// TIA Portal project "FactoryIO_Template_S7-1200_V15_V17" (V17)
// Vorlageprojekt für das Buch mit Zielsystem S7-1200

(* hardware
DEVICE "S7-1200-Station_1"  S7-1200 Station
   slot 0: "Baugruppenträger_0"  Rack  V1.0
   slot 1: "PLC_1"  CPU 1211C DC/DC/DC  6ES7 211-1AE40-0XB0  V4.1
*)

// ===== PLC "PLC_1"  CPU 1211C DC/DC/DC =====

VAR_GLOBAL   // PLC tag table "Inputs"
   "start_button" AT %I0.0 : Bool;
   "stop_button" AT %I0.1 : Bool;
   "reset_counters_button" AT %I0.2 : Bool;
   "blue_vision_sensor" AT %I0.3 : Bool;
   "green_vision_sensor" AT %I0.4 : Bool;
   "blue_count_sensor" AT %I0.5 : Bool;
   "green_count_sensor" AT %I0.6 : Bool;
   "metal_count_sensor" AT %I0.7 : Bool;
   "safety_door" AT %I1.0 : Bool;
   "emergency_stop" AT %I1.1 : Bool;
END_VAR

VAR_GLOBAL   // PLC tag table "Outputs"
   "main_conveyor" AT %Q0.0 : Bool;
   "conveyor1(blue)" AT %Q0.1 : Bool;
   "conveyor2(green)" AT %Q0.2 : Bool;
   "conveyor3(else)" AT %Q0.3 : Bool;
   "curved_conveyor" AT %Q0.4 : Bool;
   "blue_pusher" AT %Q0.5 : Bool;
   "green_pusher" AT %Q0.6 : Bool;
   "emitter" AT %Q0.7 : Bool;
   "blue_dispatch_pusher" AT %Q1.0 : Bool;
   "blue_reset" AT %Q1.1 : Bool;
   "green_dispatch_pusher" AT %Q1.2 : Bool;
   "green_reset" AT %Q1.3 : Bool;
   "metal_dispatch_pusher" AT %Q1.4 : Bool;
   "metal_reset" AT %Q1.5 : Bool;
   "alarm_siren" AT %Q1.6 : Bool;
   "warning_light" AT %Q1.7 : Bool;
   "start_light" AT %Q2.0 : Bool;
   "stop_light" AT %Q2.1 : Bool;
   "factoryIo_reset" AT %Q2.2 : Bool;
END_VAR

VAR_GLOBAL   // PLC tag table "Memory"
   "system" AT %M0.0 : Bool;
   "blue_current_value" AT %MW1 : Word;
   "green_current_value" AT %MW2 : Word;
   "metal_current_value" AT %MW3 : Word;
END_VAR

// folder: System blocks/Program resources

DATA_BLOCK "blue_counter"   // DB1
{ S7_Optimized_Access := 'TRUE' }
AUTHOR : Simatic
FAMILY : IEC
NAME : CNTR
VERSION : 1.0
// stored: InstanceOfName IEC_COUNTER
"IEC_COUNTER"
BEGIN
END_DATA_BLOCK

DATA_BLOCK "blue_delay"   // DB2
{ S7_Optimized_Access := 'TRUE' }
AUTHOR : Simatic
FAMILY : IEC
NAME : IEC_TMR
VERSION : 1.0
// stored: InstanceOfName IEC_TIMER
"IEC_TIMER"
BEGIN
END_DATA_BLOCK

DATA_BLOCK "IEC_Timer_0_DB"   // DB3
{ S7_Optimized_Access := 'TRUE' }
AUTHOR : Simatic
FAMILY : IEC
NAME : IEC_TMR
VERSION : 1.0
// stored: InstanceOfName IEC_TIMER
"IEC_TIMER"
BEGIN
END_DATA_BLOCK

DATA_BLOCK "green_counter"   // DB4
{ S7_Optimized_Access := 'TRUE' }
AUTHOR : Simatic
FAMILY : IEC
NAME : CNTR
VERSION : 1.0
// stored: InstanceOfName IEC_COUNTER
"IEC_COUNTER"
BEGIN
END_DATA_BLOCK

DATA_BLOCK "green_delay"   // DB5
{ S7_Optimized_Access := 'TRUE' }
AUTHOR : Simatic
FAMILY : IEC
NAME : IEC_TMR
VERSION : 1.0
// stored: InstanceOfName IEC_TIMER
"IEC_TIMER"
BEGIN
END_DATA_BLOCK

DATA_BLOCK "IEC_Timer_0_DB_1"   // DB6
{ S7_Optimized_Access := 'TRUE' }
AUTHOR : Simatic
FAMILY : IEC
NAME : IEC_TMR
VERSION : 1.0
// stored: InstanceOfName IEC_TIMER
"IEC_TIMER"
BEGIN
END_DATA_BLOCK

DATA_BLOCK "metal_counter"   // DB7
{ S7_Optimized_Access := 'TRUE' }
AUTHOR : Simatic
FAMILY : IEC
NAME : CNTR
VERSION : 1.0
// stored: InstanceOfName IEC_COUNTER
"IEC_COUNTER"
BEGIN
END_DATA_BLOCK

DATA_BLOCK "metal_delay"   // DB8
{ S7_Optimized_Access := 'TRUE' }
AUTHOR : Simatic
FAMILY : IEC
NAME : IEC_TMR
VERSION : 1.0
// stored: InstanceOfName IEC_TIMER
"IEC_TIMER"
BEGIN
END_DATA_BLOCK

DATA_BLOCK "IEC_Timer_0_DB_2"   // DB9
{ S7_Optimized_Access := 'TRUE' }
AUTHOR : Simatic
FAMILY : IEC
NAME : IEC_TMR
VERSION : 1.0
// stored: InstanceOfName IEC_TIMER
"IEC_TIMER"
BEGIN
END_DATA_BLOCK

// folder: (top level)

FUNCTION "MHJ-PLC-Lab-Function-S71200" : Void   // FC9000, SCL
{ S7_Optimized_Access := 'TRUE' }
VERSION : 0.1
   VAR_TEMP
      rdTimeReturn : Int;
      outputTime : DTL;
      SyncVal : Byte;
      forVal : Int;
      forVal_2 : Int;
      Value : Byte;
   END_VAR
   VAR CONSTANT
      CompVal : Byte := 16#34;
      Value_01 : Byte := 16#11;
      Value_01_DW : DWord := 16#A165_D992;
      Value_02_DW : DWord := 16#58BE_4401;
   END_VAR
BEGIN

   #Value:=PEEK(area := 16#82,
        dbNumber := 0,
        byteOffset := 511);
   #Value := #Value + 1;

   POKE(area := 16#82,
        dbNumber := 0,
        byteOffset := 511,
        value := #Value);

   POKE(area:=16#81,
        dbNumber:=0,
        byteOffset:=1016,
        value:=#Value_01_DW);
   POKE(area := 16#81,
        dbNumber := 0,
        byteOffset := 1020,
        value := #Value_02_DW);

   POKE(area := 16#81,
        dbNumber := 0,
        byteOffset := 511,
        value := B#16#00);

   FOR #forVal := 0 TO 120 DO
       FOR #forVal_2:=0 TO 10 DO
           #rdTimeReturn:=RD_SYS_T(#outputTime);
           #rdTimeReturn := WR_SYS_T(#outputTime);
           #rdTimeReturn := RD_SYS_T(#outputTime);
           #rdTimeReturn := WR_SYS_T(#outputTime);
       END_FOR;
       #SyncVal:= PEEK(area := 16#81,
                      dbNumber := 0,
                      byteOffset := 511);
       IF #SyncVal = #CompVal THEN
          GOTO M_1;
       END_IF;
   END_FOR;
   RETURN;

   M_1:
   POKE(area := 16#81,
        dbNumber := 0,
        byteOffset := 511,
        value := B#16#0);
END_FUNCTION

ORGANIZATION_BLOCK "Main"   // OB1, LAD, ProgramCycle
TITLE = "Main Program Sweep (Cycle)"
{ S7_Optimized_Access := 'TRUE' }
VERSION : 0.1
   VAR_INPUT
      Initial_Call : Bool;   // Initial call of this OB
      Remanence : Bool;   // =True, if remanent data are available
   END_VAR
BEGIN

REGION Network 1: Konnektierungsbaustein für PLC-Lab
   // Im Netzwerk 1 wird der Konnektierungsbaustein für PLC-Lab aufgerufen.
   // Dieser Aufruf darf nicht entfernt werden!
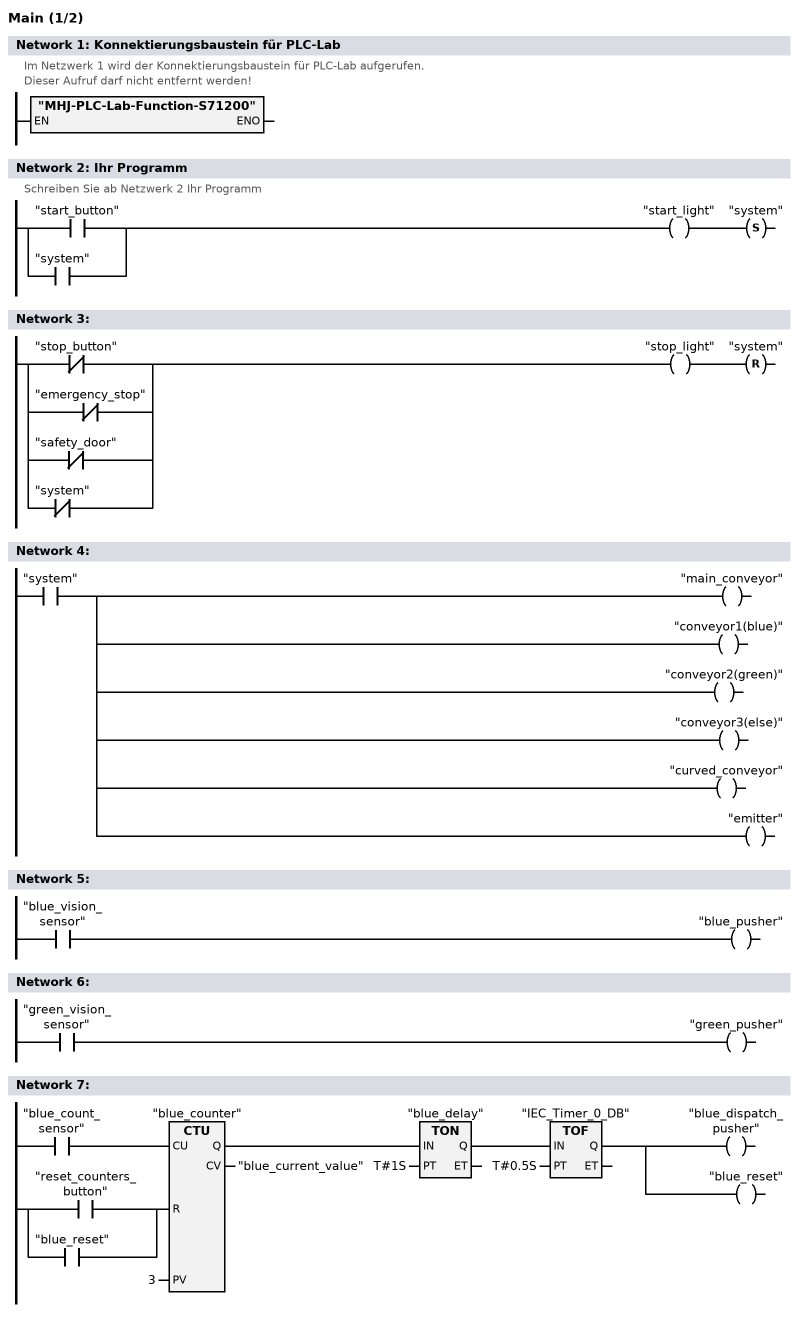
   RUNG wire#powerrail
      "MHJ-PLC-Lab-Function-S71200"()
   END_RUNG
   // the same network as SCL:
   "MHJ-PLC-Lab-Function-S71200"();
END_REGION

REGION Network 2: Ihr Programm
   // Schreiben Sie ab Netzwerk 2 Ihr Programm
   RUNG wire#powerrail
      Contact( "start_button" )
      wire#w1
      Coil( "start_light" )
      S_Coil( "system" )
   END_RUNG
   RUNG wire#powerrail
      Contact( "system" )
   END_RUNG wire#w1
   // the same network as SCL:
   "start_light" := "start_button" OR "system";
   IF "start_light" THEN "system" := TRUE; END_IF;
END_REGION

REGION Network 3
   RUNG wire#powerrail
      I_Contact( "stop_button" )
      wire#w1
      Coil( "stop_light" )
      R_Coil( "system" )
   END_RUNG
   RUNG wire#powerrail
      I_Contact( "emergency_stop" )
   END_RUNG wire#w1
   RUNG wire#powerrail
      I_Contact( "safety_door" )
   END_RUNG wire#w1
   RUNG wire#powerrail
      I_Contact( "system" )
   END_RUNG wire#w1
   // the same network as SCL:
   "stop_light" := NOT "stop_button" OR NOT "emergency_stop" OR NOT "safety_door" OR NOT "system";
   IF "stop_light" THEN "system" := FALSE; END_IF;
END_REGION

REGION Network 4
   RUNG wire#powerrail
      Contact( "system" )
      wire#w1
      Coil( "main_conveyor" )
   END_RUNG
   RUNG wire#w1
      Coil( "conveyor1(blue)" )
   END_RUNG
   RUNG wire#w1
      Coil( "conveyor2(green)" )
   END_RUNG
   RUNG wire#w1
      Coil( "conveyor3(else)" )
   END_RUNG
   RUNG wire#w1
      Coil( "curved_conveyor" )
   END_RUNG
   RUNG wire#w1
      Coil( "emitter" )
   END_RUNG
   // the same network as SCL:
   "main_conveyor" := "system";
   "conveyor1(blue)" := "system";
   "conveyor2(green)" := "system";
   "conveyor3(else)" := "system";
   "curved_conveyor" := "system";
   "emitter" := "system";
END_REGION

REGION Network 5
   RUNG wire#powerrail
      Contact( "blue_vision_sensor" )
      Coil( "blue_pusher" )
   END_RUNG
   // the same network as SCL:
   "blue_pusher" := "blue_vision_sensor";
END_REGION

REGION Network 6
   RUNG wire#powerrail
      Contact( "green_vision_sensor" )
      Coil( "green_pusher" )
   END_RUNG
   // the same network as SCL:
   "green_pusher" := "green_vision_sensor";
END_REGION

REGION Network 7
   "blue_counter".CTU(CU := "blue_count_sensor",
                      R := "reset_counters_button" OR "blue_reset",
                      PV := 3,
                      CV => "blue_current_value");
   "blue_delay".TON(IN := "blue_counter".Q, PT := T#1S);
   "IEC_Timer_0_DB".TOF(IN := "blue_delay".Q, PT := T#0.5S);
   "blue_dispatch_pusher" := "IEC_Timer_0_DB".Q;
   "blue_reset" := "IEC_Timer_0_DB".Q;
END_REGION

REGION Network 8
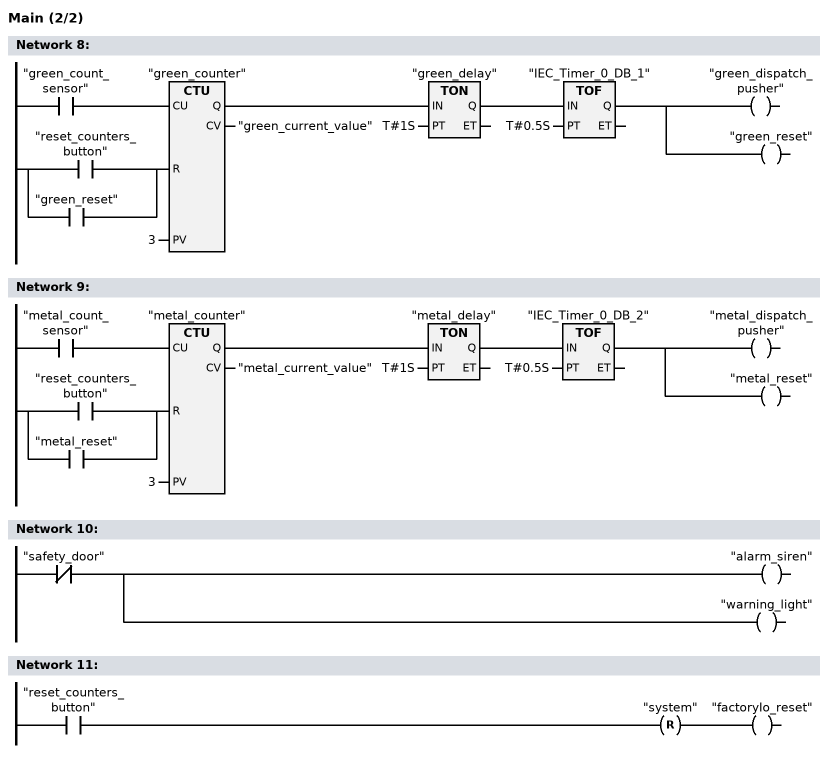
   "green_counter".CTU(CU := "green_count_sensor",
                       R := "reset_counters_button" OR "green_reset",
                       PV := 3,
                       CV => "green_current_value");
   "green_delay".TON(IN := "green_counter".Q, PT := T#1S);
   "IEC_Timer_0_DB_1".TOF(IN := "green_delay".Q, PT := T#0.5S);
   "green_dispatch_pusher" := "IEC_Timer_0_DB_1".Q;
   "green_reset" := "IEC_Timer_0_DB_1".Q;
END_REGION

REGION Network 9
   "metal_counter".CTU(CU := "metal_count_sensor",
                       R := "reset_counters_button" OR "metal_reset",
                       PV := 3,
                       CV => "metal_current_value");
   "metal_delay".TON(IN := "metal_counter".Q, PT := T#1S);
   "IEC_Timer_0_DB_2".TOF(IN := "metal_delay".Q, PT := T#0.5S);
   "metal_dispatch_pusher" := "IEC_Timer_0_DB_2".Q;
   "metal_reset" := "IEC_Timer_0_DB_2".Q;
END_REGION

REGION Network 10
   RUNG wire#powerrail
      I_Contact( "safety_door" )
      wire#w1
      Coil( "alarm_siren" )
   END_RUNG
   RUNG wire#w1
      Coil( "warning_light" )
   END_RUNG
   // the same network as SCL:
   "alarm_siren" := NOT "safety_door";
   "warning_light" := NOT "safety_door";
END_REGION

REGION Network 11
   RUNG wire#powerrail
      Contact( "reset_counters_button" )
      R_Coil( "system" )
      Coil( "factoryIo_reset" )
   END_RUNG
   // the same network as SCL:
   IF "reset_counters_button" THEN "system" := FALSE; END_IF;
   "factoryIo_reset" := "reset_counters_button";
END_REGION
END_ORGANIZATION_BLOCK